FUNCTION_BLOCK basic (* Template for a Basic Function Block Type *)
  (* Standard: 61499-2 *)
  (* Version 1.0, 2023-11-30, franz *)
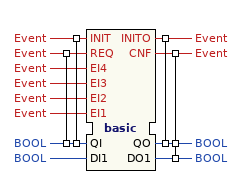
  EVENT_INPUT
    INIT WITH QI; (* Initialization Request *)
    REQ WITH QI; (* Normal Execution Request *)
    EI4;
    EI3;
    EI2;
    EI1;
  END_EVENT
  EVENT_OUTPUT
    INITO WITH QO; (* Initialization Confirm *)
    CNF WITH QO, DO1; (* Execution Confirmation *)
  END_EVENT
  VAR_INPUT
    QI : BOOL; (* Input event qualifier *)
    DI1 : BOOL;
  END_VAR
  VAR_OUTPUT
    QO : BOOL; (* Output event qualifier *)
    DO1 : BOOL;
  END_VAR
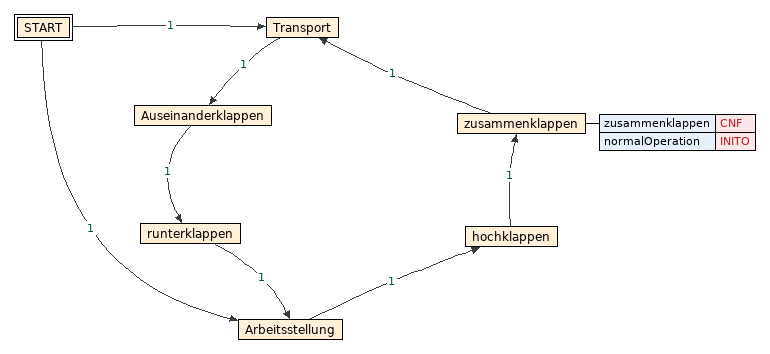
  EC_STATES
    START; (* Initial State *)
    Auseinanderklappen;
    runterklappen;
    Arbeitsstellung;
    hochklappen;
    zusammenklappen : zusammenklappen -> CNF, normalOperation -> INITO;
    Transport;
  END_STATES
  EC_TRANSITIONS
    Auseinanderklappen TO runterklappen := 1;
    runterklappen TO Arbeitsstellung := 1;
    Arbeitsstellung TO hochklappen := 1;
    hochklappen TO zusammenklappen := 1;
    Transport TO Auseinanderklappen := 1;
    zusammenklappen TO Transport := 1;
    START TO Transport := 1;
    START TO Arbeitsstellung := 1;
  END_TRANSITIONS
  ALGORITHM initialize IN ST:
QO := QI;
  END_ALGORITHM
  ALGORITHM deInitialize IN ST:
QO := FALSE;
  END_ALGORITHM
  ALGORITHM normalOperation IN ST:
QO := QI;

IF TRUE = QI THEN
	(* only perform normal operation of QI is true *)
END_IF;
  END_ALGORITHM
  ALGORITHM zusammenklappen IN ST:
QO := QI;
IF TRUE = QI THEN
	DO1 := TRUE;

END_IF;
  END_ALGORITHM
END_FUNCTION_BLOCK
